// TwinCAT 3 PLC project TcoAbstractionsTests
// Title: TcoAbstractionsTests
// Company: Vortex.Library
// ProjectVersion: 0.6.0.913
// ProgramVersion: 3.1.4024.12
// libraries:
//   Tc2_Standard, * (Beckhoff Automation GmbH)
//   Tc2_System, * (Beckhoff Automation GmbH)
//   Tc3_Module, * (Beckhoff Automation GmbH)
//   TcoAbstractions, 0.6.0.913 (Vortex.Library)
//   TcoCore, 0.6.0.913 (Vortex.Library)
// project tree:
//   / MAIN.TcPOU, PlcTask.TcTTO
// (motion and I/O tree: see PLC project tcoabstractions)
// real-time tasks:
//   TASK PlcTask: cycle T#10ms, priority 20, ADS port 350
//   TASK PlcTask1: cycle T#10ms, priority 21, ADS port 351

CONFIGURATION TcoAbstractionsTests
    RESOURCE PLC ON TwinCAT3
        TASK PlcTask(INTERVAL := T#10ms, PRIORITY := 21);
        PROGRAM MAIN WITH PlcTask : MAIN;
    END_RESOURCE
END_CONFIGURATION

// ---- MAIN.TcPOU
PROGRAM MAIN
VAR
END_VAR

END_PROGRAM
